// TIA Portal project "项目15" (V18)

(* hardware
DEVICE "S7-1500/ET200MP station_1"  S7-1500 station
   slot 0: "导轨_0"  Rack  6ES7 590-1***0-0AA0
   slot 1: "PLC_1"  CPU 1516-3 PN/DP  6ES7 516-3AN01-0AB0  V2.6
      slot 3: "CPU 显示_1"  6ES7591-1BA00-0AA0
      slot 32768: "PROFINET 接口_1"  X1
      slot 33024: "PROFINET 接口_2"  X2
      slot 33280: "DP 接口_1"  X3
   slot 2: "DI 32x24VDC HF_1"  DI 32x24VDC HF  6ES7 521-1BL00-0AB0  V2.1
   slot 3: "DQ 32x24VDC/0.5A HF_1"  DQ 32x24VDC/0.5A HF  6ES7 522-1BL01-0AB0  V1.1
   slot 4: "AI 8xU/I/RTD/TC ST_1"  AI 8xU/I/RTD/TC ST  6ES7 531-7KF00-0AB0  V2.2
   slot 5: "AQ 4xU/I ST_1"  AQ 4xU/I ST  6ES7 532-5HD00-0AB0  V2.2
DEVICE "HMI_1"  TP700 Comfort
   slot 0: "HMI_1"  TP700 Comfort  6AV2 124-0GC01-0AX0  15.1.0.0
   slot 1: "HMI_RT_1"  TP700 Comfort  6AV2 124-0GC01-0AX0  15.1.0.0
   slot 5: "HMI_1.IE_CP_1"  PROFINET Interface  15.0.1.0
      slot 1: "PROFINET Interface_1"  PROFINET Interface
         slot 1: "Port_1"  Port
         slot 2: "Port_2"  Port
   slot 7: "HMI_1.MPI/DP_CP_1"  MPI/DP Interface  15.0.1.0
*)

// ===== PLC "PLC_1"  CPU 1516-3 PN/DP =====

VAR_GLOBAL   // PLC tag table "默认变量表"
   "System_Byte" AT %MB1 : Byte;
   "FirstScan" AT %M1.0 : Bool;
   "DiagStatusUpdate" AT %M1.1 : Bool;
   "AlwaysTRUE" AT %M1.2 : Bool;
   "AlwaysFALSE" AT %M1.3 : Bool;
   "Clock_Byte" AT %MB0 : Byte;
   "Clock_10Hz" AT %M0.0 : Bool;
   "Clock_5Hz" AT %M0.1 : Bool;
   "Clock_2.5Hz" AT %M0.2 : Bool;
   "Clock_2Hz" AT %M0.3 : Bool;
   "Clock_1.25Hz" AT %M0.4 : Bool;
   "Clock_1Hz" AT %M0.5 : Bool;
   "Clock_0.625Hz" AT %M0.6 : Bool;
   "Clock_0.5Hz" AT %M0.7 : Bool;
   "蓝色按钮" AT %I1.0 : Bool;
   "蓝灯" AT %Q1.0 : Bool;
   "黄色按钮" AT %I1.1 : Bool;
   "黄灯" AT %Q1.1 : Bool;
   "急停按钮" AT %I1.3 : Bool;
END_VAR

ORGANIZATION_BLOCK "Main"   // OB1, LAD, ProgramCycle
TITLE = "Main Program Sweep (Cycle)"
{ S7_Optimized_Access := 'TRUE' }
VERSION : 0.1
   VAR_INPUT
      Initial_Call : Bool;   // Initial call of this OB
      Remanence : Bool;   // =True, if remanent data are available
   END_VAR
BEGIN

REGION Network 1
   // 这个代码有点冗余
   // 常闭触点一般都用输入
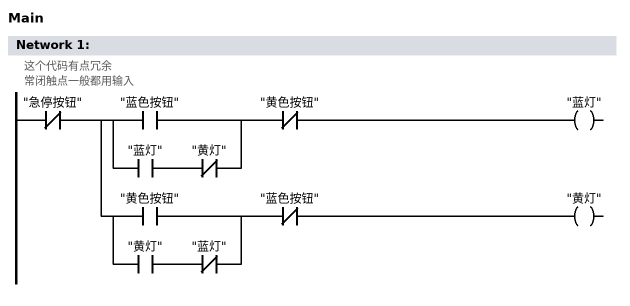
   RUNG wire#powerrail
      I_Contact( "急停按钮" )
      wire#w1
      Contact( "蓝色按钮" )
      wire#w2
      I_Contact( "黄色按钮" )
      Coil( "蓝灯" )
   END_RUNG
   RUNG wire#w1
      Contact( "蓝灯" )
      I_Contact( "黄灯" )
   END_RUNG wire#w2
   RUNG wire#w1
      Contact( "黄色按钮" )
      wire#w3
      I_Contact( "蓝色按钮" )
      Coil( "黄灯" )
   END_RUNG
   RUNG wire#w1
      Contact( "黄灯" )
      I_Contact( "蓝灯" )
   END_RUNG wire#w3
   // the same network as SCL:
   "蓝灯" := NOT "急停按钮" AND ("蓝色按钮" OR ("蓝灯" AND NOT "黄灯")) AND NOT "黄色按钮";
   "黄灯" := NOT "急停按钮" AND ("黄色按钮" OR ("黄灯" AND NOT "蓝灯")) AND NOT "蓝色按钮";
END_REGION
END_ORGANIZATION_BLOCK

(* ===== HMI "HMI_RT_1" =====
system functions are stored by id; their names below are inferred from use
connection "HMI_连接_1": ETHERNET, S7_1500_OMS

HMI tags "默认变量表"
   "Tag_ScreenNumber" : UInt, internal
   "Tag_1" : Bool = PLC 蓝色按钮 AT %I1.0, 1 s
   "Tag_3" : Bool = PLC 黄色按钮 AT %I1.1, 1 s
   "Tag_4" : Bool = PLC 黄灯 AT %Q1.1, 1 s
   "Tag_2" : Bool = PLC 蓝灯 AT %Q1.0, 1 s

screen "根画面" 800x420, template "模板_1"
   on GenerateScreen: SetTag("Tag_ScreenNumber", 1)
   Button "按钮_1" at 356,93 size 96x32; TextOff 'A'
      on Release: ResetBit("Tag_3")
      on Press: SetBit("Tag_3")
   Button "按钮_2" at 356,206 size 96x32; TextOff 'B'
      on Press: SetBit("Tag_1")
      on Release: ResetBit("Tag_1")
   Circle "圆_1" at 590,87 size 48x48
      Appearance <- "Tag_4"
   Circle "圆_2" at 587,197 size 48x48
      Appearance <- "Tag_2"

Template "模板_1" 800x420
   Button "退出" at 720,360 size 78x58; TextOff '退出'; PictureOff "ExitRuntime_TP700_Comfort_TR"; PictureOn "ExitRuntime_TP700_Comfort_TR"
      on Release: StopRuntime(0)
   Button "Template_Button" at 640,360 size 78x58; TextOff 'Text'
   Button "Template_Button_1" at 560,360 size 78x58; TextOff 'Text'
   Button "Template_Button_2" at 480,360 size 78x58; TextOff 'Text'
   Button "Template_Button_3" at 400,360 size 78x58; TextOff 'Text'
   Button "Template_Button_4" at 321,360 size 78x58; TextOff 'Text'
   Button "Template_Button_5" at 241,360 size 78x58; TextOff 'Text'
   Button "Template_Button_6" at 161,360 size 78x58; TextOff 'Text'
   Button "报警" at 81,360 size 78x58; TextOff '报警'; PictureOff "AlarmDisplay_TP700_Comfort_TR"; PictureOn "AlarmDisplay_TP700_Comfort_TR"
      on Release: function_ef3f5d25("报警窗口_Unacknowledged", -1)
   Button "起始画面" at 1,360 size 78x58; TextOff '起始画面'; PictureOff "NavigateHome_TP700_Comfort_TR"; PictureOn "NavigateHome_TP700_Comfort_TR"
      on Release: ActivateScreen("根画面", 0)
*)